FUNCTION F_CompareTypeClassWithBaseLib : BOOL
VAR_INPUT
	typeClass			: __SYSTEM.TYPE_CLASS;
	baseLibraryClass	: INT;
END_VAR
VAR
END_VAR

F_CompareTypeClassWithBaseLib := UDINT_TO_INT(typeClass) = baseLibraryClass;

END_FUNCTION

(* stored: Version 1.1.0.1, ProductVersion 3.1.4024.13
   POU F_CompareTypeClassWithBaseLib: Id {85486a24-417f-00fc-34a1-95679daea182}, SpecialFunc None *)
